{attribute 'linkalways'} 
{attribute 'no_explicit_call' := 'This FB is a CLASS and must be accessed using methods or properties'}
{attribute 'enable_dynamic_creation'}
FUNCTION_BLOCK FINAL MIN_LINT EXTENDS Node
VAR
	in1 : _LINT(0);
	in2 : _LINT(0);
	out : _LINT(0);
END_VAR

METHOD PUBLIC Clone : I_Node
VAR
	pNode : POINTER TO MIN_LINT;
END_VAR
pNode := __NEW(MIN_LINT);
Clone := pNode^;
END_METHOD

METHOD FB_init : BOOL
VAR_INPUT
	bInitRetains : BOOL; // if TRUE, the retain variables are initialized (warm start / cold start)
	bInCopyCode : BOOL;  // if TRUE, the instance afterwards gets moved into the copy code (online change)
END_VAR
AddInput('in1',THIS^.in1);
AddInput('in2',THIS^.in2);
AddOutput('out', THIS^.out);
END_METHOD

METHOD PROTECTED OnExecute
VAR
END_VAR
out.Value := MIN(in1.Value, in2.Value);
END_METHOD

END_FUNCTION_BLOCK

(* stored: Version 1.1.0.1, ProductVersion 3.1.4024.15
   POU MIN_LINT: Id {57ed9d9c-eedc-44dc-901c-176dd33140b6}, SpecialFunc None
   Folder Constructor: Id {1cb41454-59e7-4f75-82f9-e5d166e8f7a5}
   Method Clone: Id {9006a5af-bfcc-4149-9757-b130c9a2df98}
   Method FB_init: Id {59a9f51f-d349-4dce-888b-3445d6065f27}
   Method OnExecute: Id {aa0a8388-830c-456f-bc8c-2f440e0d3095} *)
